(* IEC 61131-3 sources: Elmo_Master/Lasal_PRG/Elmo_EtherCAT_Test_4Axis/Class/LMCControlCommandService (part 7) *)

	preemptRootValid :=
		(OwnershipPreemptedIdentityState[
		 LMC_OWNER_PREEMPT_HEADER_BASE]$UDINT =
		 LMC_OWNER_PREEMPT_IDENTITY_MAGIC) &
		(OwnershipPreemptedIdentityState[
		 LMC_OWNER_PREEMPT_HEADER_BASE + 2]$UDINT = AdmissionToken) &
		(OwnershipPreemptedIdentityState[
		 LMC_OWNER_PREEMPT_HEADER_BASE + 3]$UDINT = OwnerGeneration) &
		(OwnershipPreemptedIdentityState[
		 LMC_OWNER_PREEMPT_HEADER_BASE + 4]$UDINT = AxisMask) &
		(OwnershipPreemptedIdentityState[
		 LMC_OWNER_PREEMPT_HEADER_BASE + 5]$UDINT = expectedSession) &
		(OwnershipPreemptedIdentityState[
		 LMC_OWNER_PREEMPT_HEADER_BASE + 6]$UDINT = expectedSequence) &
		(OwnershipPreemptedIdentityState[
		 LMC_OWNER_PREEMPT_HEADER_BASE + 7]$UDINT =
		 (TO_UDINT(expectedCommandId) or
		  (TO_UDINT(expectedReference) shl 16))) &
		((OwnershipPreemptedIdentityState[
		  LMC_OWNER_PREEMPT_HEADER_BASE + 1]$UDINT and 0x0000FFFF) =
		 LMC_OWNER_IDENTITY_VERSION) &
		((OwnershipPreemptedIdentityState[
		  LMC_OWNER_PREEMPT_HEADER_BASE + 1]$UDINT and 0xFFFE0000) = 0);
	if (expectedAdmissionMode = LMC_OWNER_ADMISSION_SAFETY) &
	   (OwnershipPreemptedIdentityState[
	    LMC_OWNER_PREEMPT_HEADER_BASE]$UDINT =
	    LMC_OWNER_PREEMPT_IDENTITY_MAGIC) &
	   (preemptRootValid = FALSE) then
		OwnershipState[24] := 1;
		Result := -3;
		RETURN;
	end_if;
	if (expectedAdmissionMode = LMC_OWNER_ADMISSION_SAFETY) &
	   (preemptRootValid = FALSE) then
		preemptBankValid := TRUE;
		identityIndex := 0;
		while identityIndex <= 323 do
			if OwnershipPreemptedState[identityIndex] <> 0 then
				preemptBankValid := FALSE;
			end_if;
			identityIndex += 1;
		end_while;
		identityIndex := 0;
		while identityIndex <= 431 do
			if OwnershipPreemptedIdentityState[identityIndex] <> 0 then
				preemptBankValid := FALSE;
			end_if;
			identityIndex += 1;
		end_while;
		if preemptBankValid = FALSE then
			OwnershipState[24] := 1;
			Result := -3;
			RETURN;
		end_if;
	end_if;
	preemptFlags := 0;
	cleanupRequiredMask := 0;
	cleanupCompleteMask := 0;
	if preemptRootValid then
		preemptFlags := OwnershipPreemptedIdentityState[
			LMC_OWNER_PREEMPT_HEADER_BASE + 1]$UDINT;
		cleanupRequiredMask := OwnershipPreemptedIdentityState[
			LMC_OWNER_PREEMPT_HEADER_BASE + 8]$UDINT;
		cleanupCompleteMask := OwnershipPreemptedIdentityState[
			LMC_OWNER_PREEMPT_HEADER_BASE + 9]$UDINT;
		if ((cleanupRequiredMask and (not AxisMask)) <> 0) |
		   ((cleanupCompleteMask and (not cleanupRequiredMask)) <> 0) then
			OwnershipState[24] := 1;
			Result := -3;
			RETURN;
		end_if;
		preemptBankValid := TRUE;
		preemptLmcFound := FALSE;
		preemptDs402Found := FALSE;
		preemptEncoderFound := FALSE;
		axisIndex := 1;
		while axisIndex <= LMC_OWNER_AXIS_COUNT do
			case axisIndex of
				1: axisBit := 0x00000001;
				2: axisBit := 0x00000002;
				3: axisBit := 0x00000004;
				4: axisBit := 0x00000008;
				5: axisBit := 0x00000010;
				6: axisBit := 0x00000020;
				7: axisBit := 0x00000040;
				8: axisBit := 0x00000080;
				9: axisBit := 0x00000100;
			else
				axisBit := 0;
			end_case;
			preemptRecordBase := (axisIndex - 1) * LMC_OWNER_AXIS_STRIDE;
			if (OwnershipPreemptedState[preemptRecordBase] <> axisIndex) |
			   (OwnershipPreemptedState[preemptRecordBase + 35]$UDINT <>
			    (LMC_OWNER_AXIS_RECORD_MAGIC + TO_UDINT(axisIndex))) then
				preemptBankValid := FALSE;
			end_if;
			if (AxisMask and axisBit) <> 0 then
				preemptState := OwnershipPreemptedState[preemptRecordBase + 1];
				preemptOwnerKind :=
					OwnershipPreemptedState[preemptRecordBase + 2];
				preemptCommand := OwnershipPreemptedState[preemptRecordBase + 3];
				preemptToken :=
					OwnershipPreemptedState[preemptRecordBase + 4]$UDINT;
				preemptGeneration :=
					OwnershipPreemptedState[preemptRecordBase + 5]$UDINT;
				preemptSession :=
					OwnershipPreemptedState[preemptRecordBase + 6]$UDINT;
				preemptSequence :=
					OwnershipPreemptedState[preemptRecordBase + 7]$UDINT;
				preemptMask :=
					OwnershipPreemptedState[preemptRecordBase + 11]$UDINT;
				preemptReference :=
					OwnershipPreemptedState[preemptRecordBase + 12];
				preemptResourceKind :=
					OwnershipPreemptedState[preemptRecordBase + 13];
				preemptAdmission :=
					OwnershipPreemptedState[preemptRecordBase + 14];
				preemptIdentitySize :=
					OwnershipPreemptedState[preemptRecordBase + 15]$UDINT;
				preemptSpecialValid := FALSE;
				case preemptOwnerKind of
					LMC_OWNER_KIND_LMC_HOME:
						preemptSpecialValid :=
							(preemptCommand = 0x7D13) &
							(preemptResourceKind =
							 LMC_OWNER_RESOURCE_LMC_HOME_ENGINE) &
							(preemptAdmission =
							 LMC_OWNER_ADMISSION_LIFECYCLE) &
							((preemptState = LMC_OWNER_STATE_RESERVED) |
							 (preemptState =
							  LMC_OWNER_STATE_LMC_HOME_ACTIVE)) &
							(preemptIdentitySize = 56);
					LMC_OWNER_KIND_DS402_HOME:
						preemptSpecialValid :=
							(preemptCommand = 0x7D15) &
							(preemptResourceKind =
							 LMC_OWNER_RESOURCE_DS402_HOME_ENGINE) &
							(preemptAdmission =
							 LMC_OWNER_ADMISSION_LIFECYCLE) &
							((preemptState = LMC_OWNER_STATE_RESERVED) |
							 (preemptState =
							  LMC_OWNER_STATE_DS402_HOME_ACTIVE)) &
							(preemptIdentitySize = 72);
					LMC_OWNER_KIND_ENCODER:
						preemptSpecialValid :=
							(preemptCommand = 0x7E53) &
							(preemptResourceKind =
							 LMC_OWNER_RESOURCE_DIAGNOSTICS_SDO_ENGINE) &
							(preemptAdmission =
							 LMC_OWNER_ADMISSION_LIFECYCLE) &
							((preemptState = LMC_OWNER_STATE_RESERVED) |
							 (preemptState = LMC_OWNER_STATE_TW20_QUEUED) |
							 (preemptState = LMC_OWNER_STATE_TW20_RUNNING) |
							 (preemptState = LMC_OWNER_STATE_TW20_DRAINING)) &
							(preemptIdentitySize = 72);
				else
				end_case;
				if preemptSpecialValid then
					case preemptResourceKind of
						LMC_OWNER_RESOURCE_LMC_HOME_ENGINE:
							if preemptLmcFound then
								preemptBankValid := FALSE;
							end_if;
							preemptLmcFound := TRUE;
						LMC_OWNER_RESOURCE_DS402_HOME_ENGINE:
							if preemptDs402Found then
								preemptBankValid := FALSE;
							end_if;
							preemptDs402Found := TRUE;
						LMC_OWNER_RESOURCE_DIAGNOSTICS_SDO_ENGINE:
							if preemptEncoderFound then
								preemptBankValid := FALSE;
							end_if;
							preemptEncoderFound := TRUE;
					else
						preemptBankValid := FALSE;
					end_case;
					if (preemptToken = 0) | (preemptGeneration = 0) |
					   (preemptSession = 0) | (preemptSequence = 0) |
					   (preemptMask <> axisBit) |
					   (preemptReference <> axisIndex) |
					   ((cleanupRequiredMask and axisBit) = 0) then
						preemptBankValid := FALSE;
					end_if;
					if (cleanupCompleteMask and axisBit) = 0 then
						case preemptResourceKind of
							LMC_OWNER_RESOURCE_LMC_HOME_ENGINE:
								preemptBankValid := preemptBankValid &
									(OwnershipState[7]$UDINT = preemptToken) &
									(OwnershipState[8]$UDINT =
									 preemptGeneration) &
									(OwnershipState[9]$UDINT = axisBit);
							LMC_OWNER_RESOURCE_DS402_HOME_ENGINE:
								preemptBankValid := preemptBankValid &
									(OwnershipState[10]$UDINT = preemptToken) &
									(OwnershipState[11]$UDINT =
									 preemptGeneration) &
									(OwnershipState[12]$UDINT = axisBit);
							LMC_OWNER_RESOURCE_DIAGNOSTICS_SDO_ENGINE:
								preemptBankValid := preemptBankValid &
									(OwnershipState[13]$UDINT = preemptToken) &
									(OwnershipState[14]$UDINT =
									 preemptGeneration) &
									(OwnershipState[15]$UDINT = axisBit);
						else
							preemptBankValid := FALSE;
						end_case;
					else
						singletonToken := 0;
						singletonGeneration := 0;
						singletonMask := 0;
						case preemptResourceKind of
							LMC_OWNER_RESOURCE_LMC_HOME_ENGINE:
								singletonToken := OwnershipState[7]$UDINT;
								singletonGeneration := OwnershipState[8]$UDINT;
								singletonMask := OwnershipState[9]$UDINT;
							LMC_OWNER_RESOURCE_DS402_HOME_ENGINE:
								singletonToken := OwnershipState[10]$UDINT;
								singletonGeneration := OwnershipState[11]$UDINT;
								singletonMask := OwnershipState[12]$UDINT;
							LMC_OWNER_RESOURCE_DIAGNOSTICS_SDO_ENGINE:
								singletonToken := OwnershipState[13]$UDINT;
								singletonGeneration := OwnershipState[14]$UDINT;
								singletonMask := OwnershipState[15]$UDINT;
						else
							preemptBankValid := FALSE;
						end_case;
						replacementValid := (singletonToken = 0) &
							(singletonGeneration = 0) & (singletonMask = 0);
						if replacementValid = FALSE then
							replacementValid :=
								(singletonToken <> 0) &
								(singletonGeneration <> 0) &
								(singletonMask <> 0) &
								(singletonMask <= LMC_OWNER_PROFILE_AXIS_MASK) &
								((singletonMask and (singletonMask - 1)) = 0) &
								(singletonToken <> preemptToken) &
								(singletonGeneration <> preemptGeneration);
							replacementFound := FALSE;
							probeAxisIndex := 1;
							while probeAxisIndex <= LMC_OWNER_AXIS_COUNT do
								case probeAxisIndex of
									1: probeAxisBit := 0x00000001;
									2: probeAxisBit := 0x00000002;
									3: probeAxisBit := 0x00000004;
									4: probeAxisBit := 0x00000008;
									5: probeAxisBit := 0x00000010;
									6: probeAxisBit := 0x00000020;
									7: probeAxisBit := 0x00000040;
									8: probeAxisBit := 0x00000080;
									9: probeAxisBit := 0x00000100;
								else
									probeAxisBit := 0;
								end_case;
								replacementRecordBase := LMC_OWNER_GLOBAL_SLOTS +
									((probeAxisIndex - 1) * LMC_OWNER_AXIS_STRIDE);
								if singletonMask = probeAxisBit then
									if replacementFound then
										replacementValid := FALSE;
									end_if;
									replacementFound := TRUE;
									replacementStateValid := FALSE;
									case preemptOwnerKind of
										LMC_OWNER_KIND_LMC_HOME:
											replacementStateValid :=
												(OwnershipState[replacementRecordBase + 1] =
												 LMC_OWNER_STATE_RESERVED) |
												(OwnershipState[replacementRecordBase + 1] =
												 LMC_OWNER_STATE_LMC_HOME_ACTIVE) |
												(OwnershipState[replacementRecordBase + 1] =
												 LMC_OWNER_STATE_QUARANTINED);
										LMC_OWNER_KIND_DS402_HOME:
											replacementStateValid :=
												(OwnershipState[replacementRecordBase + 1] =
												 LMC_OWNER_STATE_RESERVED) |
												(OwnershipState[replacementRecordBase + 1] =
												 LMC_OWNER_STATE_DS402_HOME_ACTIVE) |
												(OwnershipState[replacementRecordBase + 1] =
												 LMC_OWNER_STATE_QUARANTINED);
										LMC_OWNER_KIND_ENCODER:
											replacementStateValid :=
												(OwnershipState[replacementRecordBase + 1] =
												 LMC_OWNER_STATE_RESERVED) |
												(OwnershipState[replacementRecordBase + 1] =
												 LMC_OWNER_STATE_TW20_QUEUED) |
												(OwnershipState[replacementRecordBase + 1] =
												 LMC_OWNER_STATE_TW20_RUNNING) |
												(OwnershipState[replacementRecordBase + 1] =
												 LMC_OWNER_STATE_TW20_DRAINING) |
												(OwnershipState[replacementRecordBase + 1] =
												 LMC_OWNER_STATE_QUARANTINED);
									else
									end_case;
									replacementIdentitySize := preemptIdentitySize;
									replacementTailSize := 0;
									if replacementIdentitySize >
									   LMC_OWNER_IDENTITY_PREFIX_BYTES then
										replacementTailSize := replacementIdentitySize -
											LMC_OWNER_IDENTITY_PREFIX_BYTES;
									end_if;
									replacementTailOffset :=
										TO_UDINT(probeAxisIndex - 1) * 8;
									replacementPackedCommand :=
										TO_UDINT(preemptCommand) or
										(TO_UDINT(probeAxisIndex) shl 16);
									replacementPackedOwner :=
										TO_UDINT(preemptOwnerKind) or
										(TO_UDINT(preemptResourceKind) shl 8) or
										(TO_UDINT(LMC_OWNER_ADMISSION_LIFECYCLE) shl 16);
									replacementHeaderBase :=
										LMC_OWNER_IDENTITY_AXIS_HEADER_BASE +
										((probeAxisIndex - 1) *
										 LMC_OWNER_IDENTITY_AXIS_HEADER_STRIDE);
									replacementValid := replacementValid &
										replacementStateValid &
										(OwnershipState[replacementRecordBase] =
										 probeAxisIndex) &
										(OwnershipState[replacementRecordBase + 35]$UDINT =
										 (LMC_OWNER_AXIS_RECORD_MAGIC +
										  TO_UDINT(probeAxisIndex))) &
										(OwnershipState[replacementRecordBase + 2] =
										 preemptOwnerKind) &
										(OwnershipState[replacementRecordBase + 3] =
										 preemptCommand) &
										(OwnershipState[replacementRecordBase + 4]$UDINT =
										 singletonToken) &
										(OwnershipState[replacementRecordBase + 5]$UDINT =
										 singletonGeneration) &
										(OwnershipState[replacementRecordBase + 6]$UDINT <> 0) &
										(OwnershipState[replacementRecordBase + 7]$UDINT <> 0) &
										(OwnershipState[replacementRecordBase + 11]$UDINT =
										 singletonMask) &
										(OwnershipState[replacementRecordBase + 12] =
										 probeAxisIndex) &
										(OwnershipState[replacementRecordBase + 13] =
										 preemptResourceKind) &
										(OwnershipState[replacementRecordBase + 14] =
										 LMC_OWNER_ADMISSION_LIFECYCLE) &
										(OwnershipState[replacementRecordBase + 15]$UDINT =
										 replacementIdentitySize) &
										(OwnershipIdentityState[replacementHeaderBase]$UDINT =
										 (LMC_OWNER_IDENTITY_AXIS_MAGIC +
										  TO_UDINT(probeAxisIndex))) &
										(OwnershipIdentityState[replacementHeaderBase + 1] =
										 LMC_OWNER_IDENTITY_VERSION) &
										(OwnershipIdentityState[replacementHeaderBase + 2]$UDINT =
										 replacementIdentitySize) &
										(OwnershipIdentityState[replacementHeaderBase + 3]$UDINT =
										 singletonToken) &
										(OwnershipIdentityState[replacementHeaderBase + 4]$UDINT =
										 singletonGeneration) &
										(OwnershipIdentityState[replacementHeaderBase + 5]$UDINT =
										 singletonMask) &
										(OwnershipIdentityState[replacementHeaderBase + 6]$UDINT =
										 OwnershipState[replacementRecordBase + 6]$UDINT) &
										(OwnershipIdentityState[replacementHeaderBase + 7]$UDINT =
										 OwnershipState[replacementRecordBase + 7]$UDINT) &
										(OwnershipIdentityState[replacementHeaderBase + 8]$UDINT =
										 replacementPackedCommand) &
										(OwnershipIdentityState[replacementHeaderBase + 9]$UDINT =
										 replacementPackedOwner) &
										(OwnershipIdentityState[replacementHeaderBase + 10]$UDINT =
										 replacementTailOffset) &
										(OwnershipIdentityState[replacementHeaderBase + 11]$UDINT =
										 replacementTailSize);
									if replacementIdentitySize = 56 then
										replacementValid := replacementValid &
											(OwnershipState[replacementRecordBase + 30] = 0) &
											(OwnershipState[replacementRecordBase + 31] = 0);
									end_if;
								elsif (OwnershipState[replacementRecordBase + 4]$UDINT =
								       singletonToken) |
								      (OwnershipState[replacementRecordBase + 5]$UDINT =
								       singletonGeneration) then
									replacementValid := FALSE;
								end_if;
								probeAxisIndex += 1;
							end_while;
							replacementValid := replacementValid & replacementFound;
						end_if;
						probeAxisIndex := 1;
						while probeAxisIndex <= LMC_OWNER_AXIS_COUNT do
							replacementRecordBase := LMC_OWNER_GLOBAL_SLOTS +
								((probeAxisIndex - 1) * LMC_OWNER_AXIS_STRIDE);
							if (OwnershipState[replacementRecordBase + 4]$UDINT =
							    preemptToken) |
							   (OwnershipState[replacementRecordBase + 5]$UDINT =
							    preemptGeneration) then
								replacementValid := FALSE;
							end_if;
							probeAxisIndex += 1;
						end_while;
						if replacementValid = FALSE then
							preemptBankValid := FALSE;
						end_if;
					end_if;
					probeAxisIndex := 1;
					while probeAxisIndex <= LMC_OWNER_AXIS_COUNT do
						probeRecordBase := (probeAxisIndex - 1) *
							LMC_OWNER_AXIS_STRIDE;
						if (probeAxisIndex <> axisIndex) &
						   ((OwnershipPreemptedState[
						     probeRecordBase + 4]$UDINT = preemptToken) |
						    (OwnershipPreemptedState[
						     probeRecordBase + 5]$UDINT =
						     preemptGeneration)) then
							preemptBankValid := FALSE;
						end_if;
						probeAxisIndex += 1;
					end_while;
				elsif (cleanupRequiredMask and axisBit) <> 0 then
					preemptBankValid := FALSE;
				end_if;
			end_if;
			axisIndex += 1;
		end_while;
		if preemptBankValid = FALSE then
			OwnershipState[24] := 1;
			Result := -3;
			RETURN;
		end_if;
	end_if;
	cleanupReady := (cleanupCompleteMask and cleanupRequiredMask) =
		cleanupRequiredMask;
	forceQuarantine :=
		(preemptFlags and LMC_OWNER_PREEMPT_FLAG_FORCE_QUARANTINE) <> 0;
	axisIndex := 1;
	while axisIndex <= LMC_OWNER_AXIS_COUNT do
		case axisIndex of
			1: axisBit := 0x00000001;
			2: axisBit := 0x00000002;
			3: axisBit := 0x00000004;
			4: axisBit := 0x00000008;
			5: axisBit := 0x00000010;
			6: axisBit := 0x00000020;
			7: axisBit := 0x00000040;
			8: axisBit := 0x00000080;
			9: axisBit := 0x00000100;
		else
			axisBit := 0;
		end_case;
		if (AxisMask and axisBit) <> 0 then
			observerBase := (axisIndex - 1) * LMC_OWNER_OBSERVER_STRIDE;
			if (OwnershipObserverState[observerBase + 5]$UDINT and
			    LMC_OWNER_OBSERVER_FORCE_QUARANTINE) <> 0 then
				forceQuarantine := TRUE;
			end_if;
		end_if;
		axisIndex += 1;
	end_while;
	if (ReportKind = LMC_OWNER_REPORT_TERMINAL_SUCCESS) &
	   (expectedAdmissionMode = LMC_OWNER_ADMISSION_SAFETY) &
	   (cleanupReady = FALSE) then
		forceQuarantine := TRUE;
	end_if;
	restoreLease :=
		(ReportKind = LMC_OWNER_REPORT_TERMINAL_SUCCESS) &
		(forceQuarantine = FALSE) &
		(expectedOwnerKind = LMC_OWNER_KIND_GROUP) &
		((expectedCommandId = 0x20A4) |
		 (expectedCommandId = 0x7D22) |
		 (expectedCommandId = 0x2085));
	if restoreLease then
		// The lease header is preserved in its bank. Prove the complete exact
		// 0x2047 lease, selected records, one-byte identity, and zero suffix
		// before the first live ownership mutation.
		leaseValid :=
			(AxisMask = LMC_OWNER_PROFILE_AXIS_MASK) &
			(OwnershipLeaseIdentityState[
			 LMC_OWNER_LEASE_IDENTITY_HEADER_BASE]$UDINT =
			 LMC_OWNER_LEASE_IDENTITY_MAGIC) &
			(OwnershipLeaseIdentityState[
			 LMC_OWNER_LEASE_IDENTITY_HEADER_BASE + 1] =
			 LMC_OWNER_IDENTITY_VERSION) &
			(OwnershipLeaseIdentityState[
			 LMC_OWNER_LEASE_IDENTITY_HEADER_BASE + 2]$UDINT = 1) &
			(OwnershipLeaseIdentityState[
			 LMC_OWNER_LEASE_IDENTITY_HEADER_BASE + 3]$UDINT <> 0) &
			(OwnershipLeaseIdentityState[
			 LMC_OWNER_LEASE_IDENTITY_HEADER_BASE + 4]$UDINT <> 0) &
			(OwnershipLeaseIdentityState[
			 LMC_OWNER_LEASE_IDENTITY_HEADER_BASE + 5]$UDINT = AxisMask) &
			(OwnershipLeaseIdentityState[
			 LMC_OWNER_LEASE_IDENTITY_HEADER_BASE + 6]$UDINT <> 0) &
			(OwnershipLeaseIdentityState[
			 LMC_OWNER_LEASE_IDENTITY_HEADER_BASE + 7]$UDINT <> 0) &
			(OwnershipLeaseIdentityState[
			 LMC_OWNER_LEASE_IDENTITY_HEADER_BASE + 8]$UDINT =
			 (TO_UDINT(0x2047) or (TO_UDINT(0x0100) shl 16))) &
			(OwnershipLeaseIdentityState[
			 LMC_OWNER_LEASE_IDENTITY_HEADER_BASE + 9]$UDINT =
			 (TO_UDINT(LMC_OWNER_KIND_GROUP) or
			  (TO_UDINT(LMC_OWNER_RESOURCE_AXIS) shl 8) or
			  (TO_UDINT(LMC_OWNER_ADMISSION_ORDINARY) shl 16)));
		leaseFirstRecordBase := -1;
		axisIndex := 1;
		while axisIndex <= LMC_OWNER_AXIS_COUNT do
			case axisIndex of
				1: axisBit := 0x00000001;
				2: axisBit := 0x00000002;
				3: axisBit := 0x00000004;
				4: axisBit := 0x00000008;
				5: axisBit := 0x00000010;
				6: axisBit := 0x00000020;
				7: axisBit := 0x00000040;
				8: axisBit := 0x00000080;
				9: axisBit := 0x00000100;
			else
				axisBit := 0;
			end_case;
			leaseRecordBase := (axisIndex - 1) * LMC_OWNER_AXIS_STRIDE;
			if (OwnershipLeaseState[leaseRecordBase] <> axisIndex) |
			   (OwnershipLeaseState[leaseRecordBase + 35]$UDINT <>
			    (LMC_OWNER_AXIS_RECORD_MAGIC + TO_UDINT(axisIndex))) then
				leaseValid := FALSE;
			end_if;
			if (AxisMask and axisBit) <> 0 then
				if (OwnershipLeaseState[leaseRecordBase + 1] <>
				    LMC_OWNER_STATE_GROUP_LEASE) |
				   (OwnershipLeaseState[leaseRecordBase + 2] <>
				    LMC_OWNER_KIND_GROUP) |
				   (OwnershipLeaseState[leaseRecordBase + 3] <> 0x2047) |
				   (OwnershipLeaseState[leaseRecordBase + 4]$UDINT <>
				    OwnershipLeaseIdentityState[
				     LMC_OWNER_LEASE_IDENTITY_HEADER_BASE + 3]$UDINT) |
				   (OwnershipLeaseState[leaseRecordBase + 5]$UDINT <>
				    OwnershipLeaseIdentityState[
				     LMC_OWNER_LEASE_IDENTITY_HEADER_BASE + 4]$UDINT) |
				   (OwnershipLeaseState[leaseRecordBase + 6]$UDINT <>
				    OwnershipLeaseIdentityState[
				     LMC_OWNER_LEASE_IDENTITY_HEADER_BASE + 6]$UDINT) |
				   (OwnershipLeaseState[leaseRecordBase + 7]$UDINT <>
				    OwnershipLeaseIdentityState[
				     LMC_OWNER_LEASE_IDENTITY_HEADER_BASE + 7]$UDINT) |
				   (OwnershipLeaseState[leaseRecordBase + 11]$UDINT <> AxisMask) |
				   (OwnershipLeaseState[leaseRecordBase + 12] <> 0x0100) |
				   (OwnershipLeaseState[leaseRecordBase + 13] <>
				    LMC_OWNER_RESOURCE_AXIS) |
				   (OwnershipLeaseState[leaseRecordBase + 14] <>
				    LMC_OWNER_ADMISSION_ORDINARY) |
				   (OwnershipLeaseState[leaseRecordBase + 15]$UDINT <> 1) |
				   (OwnershipLeaseState[leaseRecordBase + 16]$UDINT <> 1) then
					leaseValid := FALSE;
				end_if;
				identityIndex := 17;
				while identityIndex <= 31 do
					if OwnershipLeaseState[leaseRecordBase + identityIndex] <> 0 then
						leaseValid := FALSE;
					end_if;
					identityIndex += 1;
				end_while;
				if leaseFirstRecordBase < 0 then
					leaseFirstRecordBase := leaseRecordBase;
				else
					identityCompareResult := _memcmp(
						ptr1:=#OwnershipLeaseState[leaseFirstRecordBase + 16],
						ptr2:=#OwnershipLeaseState[leaseRecordBase + 16], cntr:=1);
					if identityCompareResult <> 0 then
						leaseValid := FALSE;
					end_if;
				end_if;
			else
				if (OwnershipLeaseState[leaseRecordBase + 4]$UDINT =
				    OwnershipLeaseIdentityState[
				     LMC_OWNER_LEASE_IDENTITY_HEADER_BASE + 3]$UDINT) |
				   (OwnershipLeaseState[leaseRecordBase + 5]$UDINT =
				    OwnershipLeaseIdentityState[
				     LMC_OWNER_LEASE_IDENTITY_HEADER_BASE + 4]$UDINT) then
					leaseValid := FALSE;
				end_if;
				identityIndex := 1;
				while identityIndex <= 34 do
					if OwnershipLeaseState[leaseRecordBase + identityIndex] <> 0 then
						leaseValid := FALSE;
					end_if;
					identityIndex += 1;
				end_while;
			end_if;
			axisIndex += 1;
		end_while;
		identityIndex := 0;
		while identityIndex < LMC_OWNER_IDENTITY_SUFFIX_DINTS do
			if OwnershipLeaseIdentityState[identityIndex] <> 0 then
				leaseValid := FALSE;
			end_if;
			identityIndex += 1;
		end_while;
		if leaseValid = FALSE then
			OwnershipState[24] := 1;
			Result := -3;
			RETURN;
		end_if;
	end_if;
	Result := 0;
	if preemptRootValid then
		Result += 1;
	end_if;
	if forceQuarantine then
		Result += 2;
	end_if;
	if restoreLease then
		Result += 4;
	end_if;

END_FUNCTION

FUNCTION LMCControlCommandService::HandleAdminSetPosition
	VAR_INPUT
		Reference 	: UINT;
		pRequestFrame 	: ^USINT;
		RequestFrameSize 	: UDINT;
		pResponseFrame 	: ^USINT;
		ResponseCapacity 	: UDINT;
	END_VAR
	VAR_OUTPUT
		ResponseSize 	: DINT;
	END_VAR

	ResponseSize := ProcessAdminSetPositionAsync(
		Reference:=Reference,
		pRequestFrame:=pRequestFrame,
		RequestFrameSize:=RequestFrameSize,
		pResponseFrame:=pResponseFrame,
		ResponseCapacity:=ResponseCapacity);

END_FUNCTION

FUNCTION LMCControlCommandService::DispatchRequestCommand
	VAR_INPUT
		CommandId 	: UINT;
		Reference 	: UINT;
		pRequestFrame 	: ^USINT;
		RequestFrameSize 	: UDINT;
		pResponseFrame 	: ^USINT;
		ResponseCapacity 	: UDINT;
	END_VAR
	VAR_OUTPUT
		ResponseSize 	: DINT;
	END_VAR

	ResponseSize := -1;
	if (pRequestFrame = NIL) |
	   (pResponseFrame = NIL) |
	   (RequestFrameSize < 8) then
		RETURN;
	end_if;
	case CommandId of
		0x103C, 0x1042, 0x202B:
			ResponseSize := HandleRegistryCommands(
				CommandId:=CommandId, Reference:=Reference,
				pRequestFrame:=pRequestFrame, RequestFrameSize:=RequestFrameSize,
				pResponseFrame:=pResponseFrame,
				ResponseCapacity:=ResponseCapacity);
		0x2023, 0x2024, 0x2022, 0x2028,
		0x202E, 0x209F, 0x20A0, 0x20A2:
			ResponseSize := HandleAxisCommands(
				CommandId:=CommandId, Reference:=Reference,
				pRequestFrame:=pRequestFrame, RequestFrameSize:=RequestFrameSize,
				pResponseFrame:=pResponseFrame,
				ResponseCapacity:=ResponseCapacity);
		0x20D2, 0x2047, 0x2048, 0x2049, 0x204A, 0x204B,
		0x2085, 0x20A4, 0x2045, 0x2051, 0x20E7:
			ResponseSize := HandleGroupCommands(
				CommandId:=CommandId, Reference:=Reference,
				pRequestFrame:=pRequestFrame, RequestFrameSize:=RequestFrameSize,
				pResponseFrame:=pResponseFrame,
				ResponseCapacity:=ResponseCapacity);
		0x7D12:
			ResponseSize := HandleAdminSetPosition(
				Reference:=Reference,
				pRequestFrame:=pRequestFrame, RequestFrameSize:=RequestFrameSize,
				pResponseFrame:=pResponseFrame,
				ResponseCapacity:=ResponseCapacity);
		0x7D00, 0x7D10, 0x7D14, 0x7D1A,
		0x7D13, 0x7D18, 0x7D19, 0x7D20, 0x7D22:
			ResponseSize := HandleAdminCommands(
				CommandId:=CommandId, Reference:=Reference,
				pRequestFrame:=pRequestFrame, RequestFrameSize:=RequestFrameSize,
				pResponseFrame:=pResponseFrame,
				ResponseCapacity:=ResponseCapacity);
	else
		ResponseSize := -1;
	end_case;

END_FUNCTION

FUNCTION LMCControlCommandService::ProcessAdminSetPositionAsync
	VAR_INPUT
	Reference 	: UINT;
	pRequestFrame 	: ^USINT;
	RequestFrameSize 	: UDINT;
	pResponseFrame 	: ^USINT;
	ResponseCapacity 	: UDINT;
	END_VAR
	VAR_OUTPUT
	ResponseSize 	: DINT;
	END_VAR
	VAR
	adminSetPositionKey : ARRAY [0..47] OF USINT;
	adminFrozenResponse : ARRAY [0..35] OF USINT;
	adminSchemaVersion : UINT;
	adminRequestFlags : UINT;
	adminRequestId : UDINT;
	adminDiagnosticsBuild : UDINT;
	adminBootId : UDINT;
	adminMapRevision : UDINT;
	adminClientIntentId0 : UDINT;
	adminClientIntentId1 : UDINT;
	adminClientIntentId2 : UDINT;
	adminClientIntentId3 : UDINT;
	adminAxisPosition : DINT;
	adminExpectedActualPosition : DINT;
	adminExecuteToken : UDINT;
	adminDetailCode : UDINT;
	adminOwnerSession : UDINT;
	adminOwnerSequence : UDINT;
	adminResponseSocket : DINT;
	adminContextCheck : UDINT;
	adminInvokeCheck : UDINT;
	adminIdentityCompareResult : UDINT;
	adminKeyCompareResult : UDINT;
	adminPreflightState : DINT;
	adminPreflightFailure : DINT;
	adminPreflightDetail : DINT;
	adminPreflightEvidence : UDINT;
	adminInvocationValid : BOOL;
	adminPreflightValid : BOOL;
	adminPreflightRejected : BOOL;
	adminTerminalValid : BOOL;
	END_VAR
ResponseSize := -1;
adminContextCheck := 0;
adminInvokeCheck := 0;
adminIdentityCompareResult := 0;
adminKeyCompareResult := 0;
adminPreflightState := 0;
adminPreflightFailure := 0;
adminPreflightDetail := 0;
adminPreflightEvidence := 0;
adminInvocationValid := FALSE;
adminPreflightValid := FALSE;
adminPreflightRejected := FALSE;
adminTerminalValid := FALSE;
adminDetailCode := 0;
adminRequestId := 0;
_memset(dest:=#adminSetPositionKey[0], usByte:=0, cntr:=48);
_memset(dest:=#adminFrozenResponse[0], usByte:=0, cntr:=36);
if (pRequestFrame = NIL) | (pResponseFrame = NIL) |
   (ResponseCapacity < 36) then
RETURN;
end_if;
adminInvokeCheck :=
AxisSetPositionAsyncState[114]$UDINT xor
AxisSetPositionAsyncState[115]$UDINT xor
AxisSetPositionAsyncState[116]$UDINT xor
AxisSetPositionAsyncState[117]$UDINT xor
AxisSetPositionAsyncState[118]$UDINT xor
AxisSetPositionAsyncState[119]$UDINT xor
AxisSetPositionAsyncState[120]$UDINT;
adminInvocationValid :=
(AxisSetPositionAsyncState[114]$UDINT <> 0) &
(AxisSetPositionAsyncState[115]$UDINT <> 0) &
(AxisSetPositionAsyncState[116] <> 0) &
(AxisSetPositionAsyncState[117] = 0x7D12) &
(AxisSetPositionAsyncState[118] = TO_DINT(Reference)) &
(AxisSetPositionAsyncState[119]$UDINT = 0) &
(AxisSetPositionAsyncState[120]$UDINT = 0) &
(AxisSetPositionAsyncState[121]$UDINT = adminInvokeCheck);
if adminInvocationValid = FALSE then
AxisSetPositionAsyncState[1] :=
LMC_ADMIN_SET_POSITION_ASYNC_STATE_QUARANTINED;
AxisSetPositionAsyncState[31] := 2;
ResponseSize := LMC_ADMIN_SET_POSITION_QUARANTINE_CLOSE;
RETURN;
end_if;
if RequestFrameSize >= 56 then
adminSchemaVersion := (pRequestFrame + 8)^$UINT;
adminRequestFlags := (pRequestFrame + 10)^$UINT;
adminRequestId := (pRequestFrame + 12)^$UDINT;
adminDiagnosticsBuild := (pRequestFrame + 16)^$UDINT;
adminBootId := (pRequestFrame + 20)^$UDINT;
adminMapRevision := (pRequestFrame + 24)^$UDINT;
adminClientIntentId0 := (pRequestFrame + 28)^$UDINT;
adminClientIntentId1 := (pRequestFrame + 32)^$UDINT;
adminClientIntentId2 := (pRequestFrame + 36)^$UDINT;
adminClientIntentId3 := (pRequestFrame + 40)^$UDINT;
adminAxisPosition := (pRequestFrame + 44)^$DINT;
adminExpectedActualPosition := (pRequestFrame + 48)^$DINT;
adminExecuteToken := (pRequestFrame + 52)^$UDINT;
end_if;
if RequestFrameSize <> 56 then
adminDetailCode := 5;
elsif (Reference < 1) | (Reference > 4) then
adminDetailCode := 4;
elsif adminSchemaVersion <> 1 then
adminDetailCode := 1;
elsif adminRequestFlags <> 0 then
adminDetailCode := 2;
elsif adminRequestId = 0 then
adminDetailCode := 3;
elsif adminDiagnosticsBuild = 0 then
adminDetailCode := 16;
elsif adminBootId = 0 then
adminDetailCode := 17;
elsif adminMapRevision = 0 then
adminDetailCode := 18;
elsif adminDiagnosticsBuild <> LMC_ADMIN_DIAGNOSTICS_BUILD then
adminDetailCode := 16;
elsif (OwnershipState[0]$UDINT = LMC_OWNER_TABLE_MAGIC) &
      (OwnershipState[3]$UDINT <> 0) &
      (adminBootId <> OwnershipState[3]$UDINT) then
adminDetailCode := 17;
elsif adminMapRevision <> LMC_ADMIN_MAP_REVISION then
adminDetailCode := 18;
elsif (adminClientIntentId0 = 0) &
      (adminClientIntentId1 = 0) &
      (adminClientIntentId2 = 0) &
      (adminClientIntentId3 = 0) then
adminDetailCode := 9;
elsif adminExecuteToken <> 0x50544553 then
adminDetailCode := 9;
elsif (OwnershipState[0]$UDINT <> LMC_OWNER_TABLE_MAGIC) |
      (OwnershipState[3]$UDINT = 0) then
adminDetailCode := 24;
elsif LMC_ADMIN_SET_POSITION_STORE_CONFIGURED = FALSE then
adminDetailCode := 24;
elsif IsClientConnected(#SetPositionStore) <> 1 then
adminDetailCode := 24;
end_if;
if AxisSetPositionAsyncState[1] =
   LMC_ADMIN_SET_POSITION_ASYNC_STATE_IDLE then
while adminPreflightDetail <= 127 do
if ((adminPreflightDetail < 114) |
    (adminPreflightDetail > 121)) &
   (AxisSetPositionAsyncState[adminPreflightDetail] <> 0) then
adminIdentityCompareResult := 1;
end_if;
adminPreflightDetail += 1;
end_while;
if adminIdentityCompareResult <> 0 then
AxisSetPositionAsyncState[1] :=
LMC_ADMIN_SET_POSITION_ASYNC_STATE_QUARANTINED;
AxisSetPositionAsyncState[31] := 1;
ResponseSize := LMC_ADMIN_SET_POSITION_QUARANTINE_CLOSE;
RETURN;
end_if;
end_if;
if adminDetailCode <> 0 then
if AxisSetPositionAsyncState[1] <>
   LMC_ADMIN_SET_POSITION_ASYNC_STATE_IDLE then
AxisSetPositionAsyncState[1] :=
LMC_ADMIN_SET_POSITION_ASYNC_STATE_QUARANTINED;
AxisSetPositionAsyncState[31] := 2;
if adminDetailCode = 24 then
AxisSetPositionAsyncState[31] := 7;
end_if;
ResponseSize := LMC_ADMIN_SET_POSITION_QUARANTINE_CLOSE;
RETURN;
end_if;
_memset(dest:=pResponseFrame, usByte:=0, cntr:=36);
pResponseFrame^$UINT := 0;
(pResponseFrame + 2)^$UINT := 28;
(pResponseFrame + 8)^$UINT := 1;
(pResponseFrame + 12)^$UINT := 1;
(pResponseFrame + 14)^$INT := -31000;
(pResponseFrame + 16)^$UDINT := adminRequestId;
(pResponseFrame + 20)^$UDINT := adminDetailCode;
(pResponseFrame + 28)^$UINT := 1;
ResponseSize := 36;
RETURN;
end_if;
adminSetPositionKey[0]$UINT := 1;
adminSetPositionKey[2]$UINT := 1;
adminSetPositionKey[4]$UDINT := adminDiagnosticsBuild;
adminSetPositionKey[8]$UDINT := adminBootId;
adminSetPositionKey[12]$UDINT := adminMapRevision;
adminSetPositionKey[16]$UDINT := adminRequestId;
adminSetPositionKey[20]$UDINT := adminClientIntentId0;
adminSetPositionKey[24]$UDINT := adminClientIntentId1;
adminSetPositionKey[28]$UDINT := adminClientIntentId2;
adminSetPositionKey[32]$UDINT := adminClientIntentId3;
adminSetPositionKey[36]$UINT := Reference;
adminSetPositionKey[38]$UINT := 0;
adminSetPositionKey[40]$DINT := adminAxisPosition;
adminSetPositionKey[44]$DINT := adminExpectedActualPosition;
if (AxisSetPositionAsyncState[1] >=
    LMC_ADMIN_SET_POSITION_ASYNC_STATE_BEGIN_PENDING) &
   (AxisSetPositionAsyncState[1] <=
    LMC_ADMIN_SET_POSITION_ASYNC_STATE_FRESH_ARMED) &
   ((AxisSetPositionAsyncState[0]$UDINT <>
     LMC_ADMIN_SET_POSITION_ASYNC_MAGIC) |
    (AxisSetPositionAsyncState[122] <> 0) |
    (AxisSetPositionAsyncState[123] <> 0) |
    (AxisSetPositionAsyncState[124] <> 0) |
    (AxisSetPositionAsyncState[125] <> 0) |
    (AxisSetPositionAsyncState[126] <> 0) |
    (AxisSetPositionAsyncState[127] <> 0)) then
AxisSetPositionAsyncState[1] :=
LMC_ADMIN_SET_POSITION_ASYNC_STATE_QUARANTINED;
AxisSetPositionAsyncState[31] := 1;
ResponseSize := LMC_ADMIN_SET_POSITION_QUARANTINE_CLOSE;
RETURN;
end_if;
if AxisSetPositionAsyncState[1] <>
   LMC_ADMIN_SET_POSITION_ASYNC_STATE_IDLE then
adminIdentityCompareResult := _memcmp(
ptr1:=#AxisSetPositionAsyncState[32],
ptr2:=(pRequestFrame + 8), cntr:=48);
adminKeyCompareResult := _memcmp(
ptr1:=#AxisSetPositionAsyncState[44],
ptr2:=#adminSetPositionKey[0], cntr:=48);
if (adminIdentityCompareResult <> 0) |
   (adminKeyCompareResult <> 0) then
AxisSetPositionAsyncState[1] :=
LMC_ADMIN_SET_POSITION_ASYNC_STATE_QUARANTINED;
AxisSetPositionAsyncState[31] := 1;
ResponseSize := LMC_ADMIN_SET_POSITION_QUARANTINE_CLOSE;
RETURN;
end_if;
end_if;
if (AxisSetPositionAsyncState[1] >=
    LMC_ADMIN_SET_POSITION_ASYNC_STATE_OWNERSHIP_RESERVED) &
   (AxisSetPositionAsyncState[1] <=
    LMC_ADMIN_SET_POSITION_ASYNC_STATE_QUARANTINED) then
adminContextCheck :=
LMC_ADMIN_SET_POSITION_ASYNC_MAGIC xor
AxisSetPositionAsyncState[2]$UDINT xor
AxisSetPositionAsyncState[3]$UDINT xor
AxisSetPositionAsyncState[4]$UDINT xor
AxisSetPositionAsyncState[5]$UDINT xor
AxisSetPositionAsyncState[6]$UDINT xor
AxisSetPositionAsyncState[7]$UDINT xor
AxisSetPositionAsyncState[8]$UDINT xor
AxisSetPositionAsyncState[9]$UDINT xor
AxisSetPositionAsyncState[10]$UDINT xor
AxisSetPositionAsyncState[11]$UDINT xor
AxisSetPositionAsyncState[12]$UDINT xor
AxisSetPositionAsyncState[13]$UDINT xor
AxisSetPositionAsyncState[14]$UDINT;
if (AxisSetPositionAsyncState[0]$UDINT <>
    LMC_ADMIN_SET_POSITION_ASYNC_MAGIC) |
   (AxisSetPositionAsyncState[30]$UDINT <> adminContextCheck) |
   (AxisSetPositionAsyncState[122] <> 0) |
   (AxisSetPositionAsyncState[123] <> 0) |
   (AxisSetPositionAsyncState[124] <> 0) |
   (AxisSetPositionAsyncState[125] <> 0) |
   (AxisSetPositionAsyncState[126] <> 0) |
   (AxisSetPositionAsyncState[127] <> 0) then
AxisSetPositionAsyncState[1] :=
LMC_ADMIN_SET_POSITION_ASYNC_STATE_QUARANTINED;
AxisSetPositionAsyncState[31] := 1;
ResponseSize := LMC_ADMIN_SET_POSITION_QUARANTINE_CLOSE;
RETURN;
end_if;
end_if;
if (AxisSetPositionAsyncState[1] <>
    LMC_ADMIN_SET_POSITION_ASYNC_STATE_IDLE) &
   ((AxisSetPositionAsyncState[3]$UDINT <>
     AxisSetPositionAsyncState[114]$UDINT) |
    (AxisSetPositionAsyncState[4]$UDINT <>
     AxisSetPositionAsyncState[115]$UDINT) |
    (AxisSetPositionAsyncState[8] <>
     AxisSetPositionAsyncState[116]) |
    (AxisSetPositionAsyncState[11] <> TO_DINT(Reference))) then
AxisSetPositionAsyncState[1] :=
LMC_ADMIN_SET_POSITION_ASYNC_STATE_QUARANTINED;
AxisSetPositionAsyncState[31] := 2;
ResponseSize := LMC_ADMIN_SET_POSITION_QUARANTINE_CLOSE;
RETURN;
end_if;
if ((AxisSetPositionAsyncState[1] =
     LMC_ADMIN_SET_POSITION_ASYNC_STATE_OWNERSHIP_RESERVED) |
    (AxisSetPositionAsyncState[1] =
     LMC_ADMIN_SET_POSITION_ASYNC_STATE_PREFLIGHT_PENDING)) &
   (IsClientConnected(#InputLatch) <> 1) then
AxisSetPositionAsyncState[1] :=
LMC_ADMIN_SET_POSITION_ASYNC_STATE_QUARANTINED;
AxisSetPositionAsyncState[31] := 4;
ResponseSize := LMC_ADMIN_SET_POSITION_QUARANTINE_CLOSE;
RETURN;
end_if;
if (AxisSetPositionAsyncState[1] >=
    LMC_ADMIN_SET_POSITION_ASYNC_STATE_OWNERSHIP_RESERVED) &
   (AxisSetPositionAsyncState[1] <=
    LMC_ADMIN_SET_POSITION_ASYNC_STATE_OWNERSHIP_ACTIVE) &
   ((ops.tAbsolute - AxisSetPositionAsyncState[9]$UDINT)$UDINT >=
    AxisSetPositionAsyncState[10]$UDINT) then
AxisSetPositionAsyncState[1] :=
LMC_ADMIN_SET_POSITION_ASYNC_STATE_QUARANTINED;
AxisSetPositionAsyncState[31] := 3;
ResponseSize := LMC_ADMIN_SET_POSITION_QUARANTINE_CLOSE;
RETURN;
end_if;
if AxisSetPositionAsyncState[1] =
   LMC_ADMIN_SET_POSITION_ASYNC_STATE_EXECUTION_PENDING then
AxisSetPositionAsyncState[1] :=
LMC_ADMIN_SET_POSITION_ASYNC_STATE_QUARANTINED;
AxisSetPositionAsyncState[31] := 1;
ResponseSize := LMC_ADMIN_SET_POSITION_QUARANTINE_CLOSE;
RETURN;
end_if;
// LMC_ADMIN_SET_POSITION_ASYNC_BEGIN
repeat
case AxisSetPositionAsyncState[1] of
LMC_ADMIN_SET_POSITION_ASYNC_STATE_IDLE:
adminOwnerSession := AxisSetPositionAsyncState[114]$UDINT;
adminOwnerSequence := AxisSetPositionAsyncState[115]$UDINT;
adminResponseSocket := AxisSetPositionAsyncState[116];
_memset(dest:=#AxisSetPositionAsyncState[0],
usByte:=0, cntr:=512);
AxisSetPositionAsyncState[0]$UDINT :=
LMC_ADMIN_SET_POSITION_ASYNC_MAGIC;
AxisSetPositionAsyncState[3]$UDINT := adminOwnerSession;
AxisSetPositionAsyncState[4]$UDINT := adminOwnerSequence;
AxisSetPositionAsyncState[7]$UDINT :=
TO_UDINT(1) shl TO_UDINT(Reference - 1);
AxisSetPositionAsyncState[8] := adminResponseSocket;
AxisSetPositionAsyncState[10]$UDINT := 1000;
AxisSetPositionAsyncState[11] := TO_DINT(Reference);
AxisSetPositionAsyncState[12] := adminAxisPosition;
AxisSetPositionAsyncState[13] := adminExpectedActualPosition;
AxisSetPositionAsyncState[14]$UDINT := 0;
_memcpy(ptr1:=#AxisSetPositionAsyncState[32],
ptr2:=(pRequestFrame + 8), cntr:=48);
_memcpy(ptr1:=#AxisSetPositionAsyncState[44],
ptr2:=#adminSetPositionKey[0], cntr:=48);
AxisSetPositionAsyncState[1] :=
LMC_ADMIN_SET_POSITION_ASYNC_STATE_BEGIN_PENDING;
LMC_ADMIN_SET_POSITION_ASYNC_STATE_BEGIN_PENDING:
AxisSetPositionAsyncState[21] :=
SetPositionStore.BeginSetPosition(
pKey:=#AxisSetPositionAsyncState[44], KeySize:=48,
pSnapshot:=#AxisSetPositionAsyncState[56],
SnapshotCapacity:=68,
pRecordGeneration:=(#AxisSetPositionAsyncState[2])$^UDINT,
pDetailCode:=(#AxisSetPositionAsyncState[22])$^UDINT);
if AxisSetPositionAsyncState[21] = 2 then
adminKeyCompareResult := _memcmp(
ptr1:=#AxisSetPositionAsyncState[57],
ptr2:=#AxisSetPositionAsyncState[45], cntr:=44);
adminTerminalValid :=
(AxisSetPositionAsyncState[22] = 0) &
(adminKeyCompareResult = 0) &
((AxisSetPositionAsyncState[56]$UDINT = 0x00010002) |
 (AxisSetPositionAsyncState[56]$UDINT = 0x00010003)) &
 (AxisSetPositionAsyncState[72]$UDINT =
  AxisSetPositionAsyncState[2]$UDINT) &
 (AxisSetPositionAsyncState[72]$UDINT <> 0) &
 (((AxisSetPositionAsyncState[56]$UDINT = 0x00010002) &
   (AxisSetPositionAsyncState[68] =
    AxisSetPositionAsyncState[12]) &
   (AxisSetPositionAsyncState[69] = 0) &
   (AxisSetPositionAsyncState[70] = 0) &
   (AxisSetPositionAsyncState[71] = 0)) |
  ((AxisSetPositionAsyncState[56]$UDINT = 0x00010003) &
   (AxisSetPositionAsyncState[68] = 0) &
   (((AxisSetPositionAsyncState[70]$UDINT = 11) &
     (AxisSetPositionAsyncState[69]$UDINT = 0xFFFA0001) &
     (AxisSetPositionAsyncState[71]$UDINT <> 0)) |
    ((((AxisSetPositionAsyncState[70]$UDINT = 10) |
       ((AxisSetPositionAsyncState[70]$UDINT >= 12) &
        (AxisSetPositionAsyncState[70]$UDINT <= 15))) &
      (AxisSetPositionAsyncState[69]$UDINT = 0x86E80001) &
      (AxisSetPositionAsyncState[71]$UDINT = 0))))));
if adminTerminalValid = FALSE then
AxisSetPositionAsyncState[1] :=
LMC_ADMIN_SET_POSITION_ASYNC_STATE_QUARANTINED;
AxisSetPositionAsyncState[31] := 7;
ResponseSize := LMC_ADMIN_SET_POSITION_QUARANTINE_CLOSE;
RETURN;
end_if;
adminFrozenResponse[0]$UINT := 0;
adminFrozenResponse[2]$UINT := 28;
adminFrozenResponse[4]$UDINT := 0;
adminFrozenResponse[8]$UINT := 1;
adminFrozenResponse[10]$UINT := 0;
adminFrozenResponse[12]$UINT :=
AxisSetPositionAsyncState[69]$UINT;
adminFrozenResponse[14]$INT := TO_INT(
AxisSetPositionAsyncState[69]$UDINT / 65536);
adminFrozenResponse[16]$UDINT :=
AxisSetPositionAsyncState[60]$UDINT;
adminFrozenResponse[20]$UDINT :=
AxisSetPositionAsyncState[70]$UDINT;
adminFrozenResponse[24]$DINT :=
AxisSetPositionAsyncState[68];
adminFrozenResponse[28]$UINT := 1;
adminFrozenResponse[30]$UINT := 0;
adminFrozenResponse[32]$UDINT :=
AxisSetPositionAsyncState[71]$UDINT;
_memcpy(ptr1:=#AxisSetPositionAsyncState[105],
ptr2:=#adminFrozenResponse[0], cntr:=36);
_memcpy(ptr1:=pResponseFrame,
ptr2:=#AxisSetPositionAsyncState[105], cntr:=36);
_memset(dest:=#AxisSetPositionAsyncState[0],
usByte:=0, cntr:=512);
ResponseSize := 36;
RETURN;
elsif AxisSetPositionAsyncState[21] = 1 then
if (AxisSetPositionAsyncState[22] = 0) &
   (AxisSetPositionAsyncState[2]$UDINT <> 0) then
AxisSetPositionAsyncState[9]$UDINT := ops.tAbsolute;
AxisSetPositionAsyncState[1] :=
LMC_ADMIN_SET_POSITION_ASYNC_STATE_FRESH_ARMED;
else
AxisSetPositionAsyncState[1] :=
LMC_ADMIN_SET_POSITION_ASYNC_STATE_QUARANTINED;
AxisSetPositionAsyncState[31] := 7;
ResponseSize := LMC_ADMIN_SET_POSITION_QUARANTINE_CLOSE;
RETURN;
end_if;
elsif AxisSetPositionAsyncState[21] = 0 then
if (AxisSetPositionAsyncState[22] = 20) |
   (AxisSetPositionAsyncState[22] = 21) |
   (AxisSetPositionAsyncState[22] = 23) |
   (AxisSetPositionAsyncState[22] = 24) then
_memset(dest:=pResponseFrame, usByte:=0, cntr:=36);
pResponseFrame^$UINT := 0;
(pResponseFrame + 2)^$UINT := 28;
(pResponseFrame + 8)^$UINT := 1;
(pResponseFrame + 12)^$UINT := 1;
(pResponseFrame + 14)^$INT := -31000;
(pResponseFrame + 16)^$UDINT :=
AxisSetPositionAsyncState[48]$UDINT;
(pResponseFrame + 20)^$UDINT :=
AxisSetPositionAsyncState[22]$UDINT;
(pResponseFrame + 28)^$UINT := 1;
_memset(dest:=#AxisSetPositionAsyncState[0],
usByte:=0, cntr:=512);
ResponseSize := 36;
RETURN;
else
AxisSetPositionAsyncState[1] :=
LMC_ADMIN_SET_POSITION_ASYNC_STATE_QUARANTINED;
AxisSetPositionAsyncState[31] := 7;
ResponseSize := LMC_ADMIN_SET_POSITION_QUARANTINE_CLOSE;
RETURN;
end_if;
else
AxisSetPositionAsyncState[1] :=
LMC_ADMIN_SET_POSITION_ASYNC_STATE_QUARANTINED;
AxisSetPositionAsyncState[31] := 7;
ResponseSize := LMC_ADMIN_SET_POSITION_QUARANTINE_CLOSE;
RETURN;
end_if;
LMC_ADMIN_SET_POSITION_ASYNC_STATE_FRESH_ARMED:
AxisSetPositionAsyncState[24] := ReserveAxisOwnership(
CommandId:=0x7D12, Reference:=Reference,
RequestedAxisMask:=AxisSetPositionAsyncState[7]$UDINT,
OwnerKind:=LMC_OWNER_KIND_DIRECT,
ResourceKind:=LMC_OWNER_RESOURCE_AXIS,
AdmissionMode:=LMC_OWNER_ADMISSION_ORDINARY,
CallerSessionEpoch:=AxisSetPositionAsyncState[3]$UDINT,
RequestSequence:=AxisSetPositionAsyncState[4]$UDINT,
pIdentity:=(#AxisSetPositionAsyncState[32])$^void,
IdentitySize:=48,
pEffectiveAxisMask:=(#AxisSetPositionAsyncState[23])$^UDINT,
pAdmissionToken:=(#AxisSetPositionAsyncState[5])$^UDINT,
pOwnerGeneration:=(#AxisSetPositionAsyncState[6])$^UDINT);
if (AxisSetPositionAsyncState[24] = 0) &
   (AxisSetPositionAsyncState[23]$UDINT =
    AxisSetPositionAsyncState[7]$UDINT) &
   (AxisSetPositionAsyncState[5]$UDINT <> 0) &
   (AxisSetPositionAsyncState[6]$UDINT <> 0) then
AxisSetPositionAsyncState[1] :=
LMC_ADMIN_SET_POSITION_ASYNC_STATE_OWNERSHIP_RESERVED;
else
AxisSetPositionAsyncState[1] :=
LMC_ADMIN_SET_POSITION_ASYNC_STATE_QUARANTINED;
AxisSetPositionAsyncState[31] := 5;
ResponseSize := LMC_ADMIN_SET_POSITION_QUARANTINE_CLOSE;
RETURN;
end_if;
adminContextCheck :=
LMC_ADMIN_SET_POSITION_ASYNC_MAGIC xor
AxisSetPositionAsyncState[2]$UDINT xor
AxisSetPositionAsyncState[3]$UDINT xor
AxisSetPositionAsyncState[4]$UDINT xor
AxisSetPositionAsyncState[5]$UDINT xor
AxisSetPositionAsyncState[6]$UDINT xor
AxisSetPositionAsyncState[7]$UDINT xor
AxisSetPositionAsyncState[8]$UDINT xor
AxisSetPositionAsyncState[9]$UDINT xor
AxisSetPositionAsyncState[10]$UDINT xor
AxisSetPositionAsyncState[11]$UDINT xor
AxisSetPositionAsyncState[12]$UDINT xor
AxisSetPositionAsyncState[13]$UDINT xor
AxisSetPositionAsyncState[14]$UDINT;
AxisSetPositionAsyncState[30]$UDINT := adminContextCheck;
adminContextCheck :=
LMC_ADMIN_SET_POSITION_ASYNC_MAGIC xor
AxisSetPositionAsyncState[2]$UDINT xor
AxisSetPositionAsyncState[3]$UDINT xor
AxisSetPositionAsyncState[4]$UDINT xor
AxisSetPositionAsyncState[5]$UDINT xor
AxisSetPositionAsyncState[6]$UDINT xor
AxisSetPositionAsyncState[7]$UDINT xor
AxisSetPositionAsyncState[8]$UDINT xor
AxisSetPositionAsyncState[9]$UDINT xor
AxisSetPositionAsyncState[10]$UDINT xor
AxisSetPositionAsyncState[11]$UDINT xor
AxisSetPositionAsyncState[12]$UDINT xor
AxisSetPositionAsyncState[13]$UDINT xor
AxisSetPositionAsyncState[14]$UDINT;
if (AxisSetPositionAsyncState[30]$UDINT = adminContextCheck) then
ResponseSize := LMC_ADMIN_SET_POSITION_PENDING;
RETURN;
else
AxisSetPositionAsyncState[1] :=
LMC_ADMIN_SET_POSITION_ASYNC_STATE_QUARANTINED;
AxisSetPositionAsyncState[31] := 1;
ResponseSize := LMC_ADMIN_SET_POSITION_QUARANTINE_CLOSE;
RETURN;
end_if;
LMC_ADMIN_SET_POSITION_ASYNC_STATE_OWNERSHIP_RESERVED:
AxisSetPositionAsyncState[28] :=
InputLatch.SubmitAxisSetPositionPreflight(
OperationToken:=AxisSetPositionAsyncState[5]$UDINT,
OwnerGeneration:=AxisSetPositionAsyncState[6]$UDINT,
StoreRecordGeneration:=AxisSetPositionAsyncState[2]$UDINT,
CallerSessionEpoch:=AxisSetPositionAsyncState[3]$UDINT,
RequestSequence:=AxisSetPositionAsyncState[4]$UDINT,
AxisReference:=AxisSetPositionAsyncState[11],
TargetPosition:=AxisSetPositionAsyncState[12],
ExpectedActualPosition:=AxisSetPositionAsyncState[13],
MaxJump:=AxisSetPositionAsyncState[14]$UDINT,
ExpectedAxisMask:=AxisSetPositionAsyncState[7]$UDINT);
if (AxisSetPositionAsyncState[28] = 0) |
   (AxisSetPositionAsyncState[28] = 1) then
AxisSetPositionAsyncState[1] :=
LMC_ADMIN_SET_POSITION_ASYNC_STATE_PREFLIGHT_PENDING;
ResponseSize := LMC_ADMIN_SET_POSITION_PENDING;
else
AxisSetPositionAsyncState[1] :=
LMC_ADMIN_SET_POSITION_ASYNC_STATE_QUARANTINED;
AxisSetPositionAsyncState[31] := 4;
ResponseSize := LMC_ADMIN_SET_POSITION_QUARANTINE_CLOSE;
RETURN;
end_if;
RETURN;
LMC_ADMIN_SET_POSITION_ASYNC_STATE_PREFLIGHT_PENDING:
AxisSetPositionAsyncState[29] :=
InputLatch.CopyAxisSetPositionPreflightResult(
OperationToken:=AxisSetPositionAsyncState[5]$UDINT,
OwnerGeneration:=AxisSetPositionAsyncState[6]$UDINT,
StoreRecordGeneration:=AxisSetPositionAsyncState[2]$UDINT,
pDest:=#AxisSetPositionAsyncState[73], DestSize:=128);
if AxisSetPositionAsyncState[29] = 1 then
ResponseSize := LMC_ADMIN_SET_POSITION_PENDING;
RETURN;
elsif AxisSetPositionAsyncState[29] <> 0 then
AxisSetPositionAsyncState[1] :=
LMC_ADMIN_SET_POSITION_ASYNC_STATE_QUARANTINED;
AxisSetPositionAsyncState[31] := 4;
ResponseSize := LMC_ADMIN_SET_POSITION_QUARANTINE_CLOSE;
RETURN;
end_if;
adminPreflightState := AxisSetPositionAsyncState[84];
adminPreflightFailure := AxisSetPositionAsyncState[85];
adminPreflightDetail := AxisSetPositionAsyncState[86];
adminPreflightEvidence := AxisSetPositionAsyncState[101]$UDINT;
adminPreflightRejected :=
(adminPreflightState = LMC_SET_POSITION_PREFLIGHT_REJECTED) &
(((adminPreflightFailure = LMC_SET_POSITION_PREFLIGHT_CLIENT) &
  (adminPreflightDetail = 10)) |
 ((adminPreflightFailure = LMC_SET_POSITION_PREFLIGHT_STATE) &
  (adminPreflightDetail = 10)) |
 ((adminPreflightFailure = LMC_SET_POSITION_PREFLIGHT_CONFIG) &
  (adminPreflightDetail = 14)) |
 ((adminPreflightFailure = LMC_SET_POSITION_PREFLIGHT_VELOCITY) &
  (adminPreflightDetail = 12)) |
 ((adminPreflightFailure = LMC_SET_POSITION_PREFLIGHT_AXIS_ERROR) &
  (adminPreflightDetail = 13)) |
 ((adminPreflightFailure = LMC_SET_POSITION_PREFLIGHT_COORDINATE) &
  (adminPreflightDetail = 15))) &
((adminPreflightEvidence and
  LMC_SET_POSITION_EVIDENCE_REJECT_MASK) =
 LMC_SET_POSITION_EVIDENCE_REJECT_MASK);
adminPreflightValid :=
(AxisSetPositionAsyncState[73]$UDINT =
 AxisSetPositionAsyncState[5]$UDINT) &
(AxisSetPositionAsyncState[74]$UDINT =
 AxisSetPositionAsyncState[6]$UDINT) &
(AxisSetPositionAsyncState[75]$UDINT =
 AxisSetPositionAsyncState[2]$UDINT) &
(AxisSetPositionAsyncState[76]$UDINT =
 AxisSetPositionAsyncState[3]$UDINT) &
(AxisSetPositionAsyncState[77]$UDINT =
 AxisSetPositionAsyncState[4]$UDINT) &
(AxisSetPositionAsyncState[78]$UDINT =
 AxisSetPositionAsyncState[11]$UDINT) &
(AxisSetPositionAsyncState[79]$UDINT =
 AxisSetPositionAsyncState[12]$UDINT) &
(AxisSetPositionAsyncState[80]$UDINT =
 AxisSetPositionAsyncState[13]$UDINT) &
(AxisSetPositionAsyncState[81]$UDINT =
 AxisSetPositionAsyncState[14]$UDINT) &
(AxisSetPositionAsyncState[82]$UDINT =
 AxisSetPositionAsyncState[7]$UDINT) &
(AxisSetPositionAsyncState[83]$UDINT <> 0) &
((AxisSetPositionAsyncState[15]$UDINT = 0) |
 (AxisSetPositionAsyncState[83]$UDINT =
  AxisSetPositionAsyncState[15]$UDINT)) &
(AxisSetPositionAsyncState[102] = 0) &
(AxisSetPositionAsyncState[103] = 0) &
(AxisSetPositionAsyncState[104] = 0) &
(((adminPreflightState = LMC_SET_POSITION_PREFLIGHT_READY) &
  (adminPreflightFailure = 0) &
  (adminPreflightDetail = 0) &
  (adminPreflightEvidence =
   LMC_SET_POSITION_EVIDENCE_READY_MASK)) |
 adminPreflightRejected);
if adminPreflightValid = FALSE then
AxisSetPositionAsyncState[1] :=
LMC_ADMIN_SET_POSITION_ASYNC_STATE_QUARANTINED;
AxisSetPositionAsyncState[31] := 4;
ResponseSize := LMC_ADMIN_SET_POSITION_QUARANTINE_CLOSE;
RETURN;
end_if;
if AxisSetPositionAsyncState[15]$UDINT = 0 then
AxisSetPositionAsyncState[15]$UDINT :=
AxisSetPositionAsyncState[83]$UDINT;
end_if;
if adminPreflightState = LMC_SET_POSITION_PREFLIGHT_READY then
AxisSetPositionAsyncState[1] :=
LMC_ADMIN_SET_POSITION_ASYNC_STATE_PREFLIGHT_READY;
else
AxisSetPositionAsyncState[16] := adminPreflightDetail;
AxisSetPositionAsyncState[17] := 1;
AxisSetPositionAsyncState[18] := -31000;
AxisSetPositionAsyncState[19] := 0;
AxisSetPositionAsyncState[20] := 0;
AxisSetPositionAsyncState[1] :=
LMC_ADMIN_SET_POSITION_ASYNC_STATE_TERMINAL_COMMIT_PENDING;
end_if;
LMC_ADMIN_SET_POSITION_ASYNC_STATE_PREFLIGHT_READY:
adminPreflightValid :=
(AxisSetPositionAsyncState[102] = 0) &
(AxisSetPositionAsyncState[103] = 0) &
(AxisSetPositionAsyncState[104] = 0);
if adminPreflightValid = FALSE then
AxisSetPositionAsyncState[1] :=
LMC_ADMIN_SET_POSITION_ASYNC_STATE_QUARANTINED;
AxisSetPositionAsyncState[31] := 4;
ResponseSize := LMC_ADMIN_SET_POSITION_QUARANTINE_CLOSE;
RETURN;
end_if;
AxisSetPositionAsyncState[25] := ValidateAxisOwnershipIdentity(
CommandId:=0x7D12,
Reference:=AxisSetPositionAsyncState[11]$UINT,
ExpectedAxisMask:=AxisSetPositionAsyncState[7]$UDINT,
OwnerKind:=LMC_OWNER_KIND_DIRECT,
ResourceKind:=LMC_OWNER_RESOURCE_AXIS,
AdmissionMode:=LMC_OWNER_ADMISSION_ORDINARY,
CallerSessionEpoch:=AxisSetPositionAsyncState[3]$UDINT,
RequestSequence:=AxisSetPositionAsyncState[4]$UDINT,
AdmissionToken:=AxisSetPositionAsyncState[5]$UDINT,
OwnerGeneration:=AxisSetPositionAsyncState[6]$UDINT,
RequiredPhase:=LMC_OWNER_PHASE_RESERVED,
pIdentity:=#AxisSetPositionAsyncState[32],
IdentitySize:=48);
if AxisSetPositionAsyncState[25] <> 0 then
AxisSetPositionAsyncState[1] :=
LMC_ADMIN_SET_POSITION_ASYNC_STATE_QUARANTINED;
AxisSetPositionAsyncState[31] := 5;
ResponseSize := LMC_ADMIN_SET_POSITION_QUARANTINE_CLOSE;
RETURN;
end_if;
AxisSetPositionAsyncState[26] := CommitAxisOwnership(
CommandId:=0x7D12,
Reference:=AxisSetPositionAsyncState[11]$UINT,
ExpectedAxisMask:=AxisSetPositionAsyncState[7]$UDINT,
CallerSessionEpoch:=AxisSetPositionAsyncState[3]$UDINT,
RequestSequence:=AxisSetPositionAsyncState[4]$UDINT,
AdmissionToken:=AxisSetPositionAsyncState[5]$UDINT,
OwnerGeneration:=AxisSetPositionAsyncState[6]$UDINT);
if AxisSetPositionAsyncState[26] <> 0 then
AxisSetPositionAsyncState[1] :=
LMC_ADMIN_SET_POSITION_ASYNC_STATE_QUARANTINED;
AxisSetPositionAsyncState[31] := 5;
ResponseSize := LMC_ADMIN_SET_POSITION_QUARANTINE_CLOSE;
RETURN;
end_if;
AxisSetPositionAsyncState[25] := ValidateAxisOwnershipIdentity(
CommandId:=0x7D12,
Reference:=AxisSetPositionAsyncState[11]$UINT,
ExpectedAxisMask:=AxisSetPositionAsyncState[7]$UDINT,
OwnerKind:=LMC_OWNER_KIND_DIRECT,
ResourceKind:=LMC_OWNER_RESOURCE_AXIS,
AdmissionMode:=LMC_OWNER_ADMISSION_ORDINARY,
CallerSessionEpoch:=AxisSetPositionAsyncState[3]$UDINT,
RequestSequence:=AxisSetPositionAsyncState[4]$UDINT,
AdmissionToken:=AxisSetPositionAsyncState[5]$UDINT,
OwnerGeneration:=AxisSetPositionAsyncState[6]$UDINT,
RequiredPhase:=LMC_OWNER_PHASE_ACTIVE,
pIdentity:=#AxisSetPositionAsyncState[32],
IdentitySize:=48);
if AxisSetPositionAsyncState[25] <> 0 then
AxisSetPositionAsyncState[1] :=
LMC_ADMIN_SET_POSITION_ASYNC_STATE_QUARANTINED;
AxisSetPositionAsyncState[31] := 5;
ResponseSize := LMC_ADMIN_SET_POSITION_QUARANTINE_CLOSE;
RETURN;
end_if;
AxisSetPositionAsyncState[1] :=
LMC_ADMIN_SET_POSITION_ASYNC_STATE_OWNERSHIP_ACTIVE;
ResponseSize := LMC_ADMIN_SET_POSITION_PENDING;
RETURN;
LMC_ADMIN_SET_POSITION_ASYNC_STATE_OWNERSHIP_ACTIVE:
ResponseSize := LMC_ADMIN_SET_POSITION_PENDING;
RETURN;
LMC_ADMIN_SET_POSITION_ASYNC_STATE_EXECUTION_PENDING:
// P2 only.
RETURN;
LMC_ADMIN_SET_POSITION_ASYNC_STATE_TERMINAL_COMMIT_PENDING:
AxisSetPositionAsyncState[21] :=
SetPositionStore.CommitSetPositionTerminal(
pKey:=#AxisSetPositionAsyncState[44], KeySize:=48,
RecordGeneration:=AxisSetPositionAsyncState[2]$UDINT,
RecordState:=3,
AppliedPosition:=AxisSetPositionAsyncState[19],
OriginalCommandStatus:=AxisSetPositionAsyncState[17]$UINT,
OriginalErrorId:=AxisSetPositionAsyncState[18]$INT,
OriginalDetailCode:=AxisSetPositionAsyncState[16]$UDINT,
NativeCommandState:=AxisSetPositionAsyncState[20]$UDINT,
pSnapshot:=#AxisSetPositionAsyncState[56],
SnapshotCapacity:=68,
pDetailCode:=(#AxisSetPositionAsyncState[22])$^UDINT);
adminKeyCompareResult := _memcmp(
ptr1:=#AxisSetPositionAsyncState[57],
ptr2:=#AxisSetPositionAsyncState[45], cntr:=44);
adminTerminalValid :=
(AxisSetPositionAsyncState[21] = 1) &
(AxisSetPositionAsyncState[22] = 0) &
(AxisSetPositionAsyncState[56]$UDINT = 0x00010003) &
(adminKeyCompareResult = 0) &
(AxisSetPositionAsyncState[68] =
 AxisSetPositionAsyncState[19]) &
(AxisSetPositionAsyncState[69]$UDINT = 0x86E80001) &
(AxisSetPositionAsyncState[70]$UDINT =
 AxisSetPositionAsyncState[16]$UDINT) &
(AxisSetPositionAsyncState[71]$UDINT =
 AxisSetPositionAsyncState[20]$UDINT) &
(AxisSetPositionAsyncState[72]$UDINT =
 AxisSetPositionAsyncState[2]$UDINT);
if adminTerminalValid then
AxisSetPositionAsyncState[1] :=
LMC_ADMIN_SET_POSITION_ASYNC_STATE_TERMINAL_PROVEN;
elsif (AxisSetPositionAsyncState[21] = 1) |
      (AxisSetPositionAsyncState[21] =
       LMC_ADMIN_SET_POSITION_CLOSE_WITHOUT_RESPONSE) then
ResponseSize :=
LMC_ADMIN_SET_POSITION_CLOSE_WITHOUT_RESPONSE;
RETURN;
else
AxisSetPositionAsyncState[1] :=
LMC_ADMIN_SET_POSITION_ASYNC_STATE_QUARANTINED;
AxisSetPositionAsyncState[31] := 7;
ResponseSize := LMC_ADMIN_SET_POSITION_QUARANTINE_CLOSE;
RETURN;
end_if;
LMC_ADMIN_SET_POSITION_ASYNC_STATE_TERMINAL_PROVEN:
AxisSetPositionAsyncState[27] := RollbackAxisOwnership(
AdmissionToken:=AxisSetPositionAsyncState[5]$UDINT,
OwnerGeneration:=AxisSetPositionAsyncState[6]$UDINT,
CallerSessionEpoch:=AxisSetPositionAsyncState[3]$UDINT,
RequestSequence:=AxisSetPositionAsyncState[4]$UDINT,
Reason:=0);
if AxisSetPositionAsyncState[27] <> 0 then
AxisSetPositionAsyncState[1] :=
LMC_ADMIN_SET_POSITION_ASYNC_STATE_QUARANTINED;
AxisSetPositionAsyncState[31] := 6;
ResponseSize := LMC_ADMIN_SET_POSITION_QUARANTINE_CLOSE;
RETURN;
end_if;
adminFrozenResponse[0]$UINT := 0;
adminFrozenResponse[2]$UINT := 28;
adminFrozenResponse[4]$UDINT := 0;
adminFrozenResponse[8]$UINT := 1;
adminFrozenResponse[10]$UINT := 0;
adminFrozenResponse[12]$UINT :=
AxisSetPositionAsyncState[69]$UINT;
adminFrozenResponse[14]$INT := TO_INT(
AxisSetPositionAsyncState[69]$UDINT / 65536);
adminFrozenResponse[16]$UDINT :=
AxisSetPositionAsyncState[60]$UDINT;
adminFrozenResponse[20]$UDINT :=
AxisSetPositionAsyncState[70]$UDINT;
adminFrozenResponse[24]$DINT := AxisSetPositionAsyncState[68];
adminFrozenResponse[28]$UINT := 1;
adminFrozenResponse[30]$UINT := 0;
adminFrozenResponse[32]$UDINT :=
AxisSetPositionAsyncState[71]$UDINT;
_memcpy(ptr1:=#AxisSetPositionAsyncState[105],
ptr2:=#adminFrozenResponse[0], cntr:=36);
_memcpy(ptr1:=pResponseFrame,
ptr2:=#AxisSetPositionAsyncState[105], cntr:=36);
_memset(dest:=#AxisSetPositionAsyncState[0],
usByte:=0, cntr:=512);
ResponseSize := 36;
RETURN;
LMC_ADMIN_SET_POSITION_ASYNC_STATE_QUARANTINED:
ResponseSize := LMC_ADMIN_SET_POSITION_QUARANTINE_CLOSE;
RETURN;
else
AxisSetPositionAsyncState[1] :=
LMC_ADMIN_SET_POSITION_ASYNC_STATE_QUARANTINED;
AxisSetPositionAsyncState[31] := 1;
ResponseSize := LMC_ADMIN_SET_POSITION_QUARANTINE_CLOSE;
RETURN;
end_case;
until (AxisSetPositionAsyncState[1] <>
       LMC_ADMIN_SET_POSITION_ASYNC_STATE_BEGIN_PENDING) &
      (AxisSetPositionAsyncState[1] <>
       LMC_ADMIN_SET_POSITION_ASYNC_STATE_FRESH_ARMED) &
      (AxisSetPositionAsyncState[1] <>
       LMC_ADMIN_SET_POSITION_ASYNC_STATE_PREFLIGHT_READY) &
      (AxisSetPositionAsyncState[1] <>
       LMC_ADMIN_SET_POSITION_ASYNC_STATE_TERMINAL_COMMIT_PENDING) &
      (AxisSetPositionAsyncState[1] <>
       LMC_ADMIN_SET_POSITION_ASYNC_STATE_TERMINAL_PROVEN)
end_repeat;
// LMC_ADMIN_SET_POSITION_ASYNC_END
END_FUNCTION
